FUNCTION DecINT : INT				// Increments the given UINT value
VAR_IN_OUT
	ioNum:	INT;		// Value to increment
END_VAR

DecINT := ioNum := ioNum - 1;

END_FUNCTION

(* stored: Version 1.1.0.1, ProductVersion 3.1.4026.18
   POU DecINT: Id {f2d3e73d-0f4d-4120-ab2a-64f22c5f5e67}, SpecialFunc None *)
